# EPICS autosave request: iocs/qimageIOC/iocBoot/iocQImage/auto_settings.req
file "ADBase_settings.req",       P=$(P),  R=cam1:
file "qimaging_settings.req",       P=$(P),  R=cam1:
file "NDPluginBase_settings.req", P=$(P),  R=image1:
file "NDStdArrays_settings.req",  P=$(P),  R=image1:
file "commonPlugin_settings.req", P=$(P)
